RoboDK station: Drillingtask2.rdk

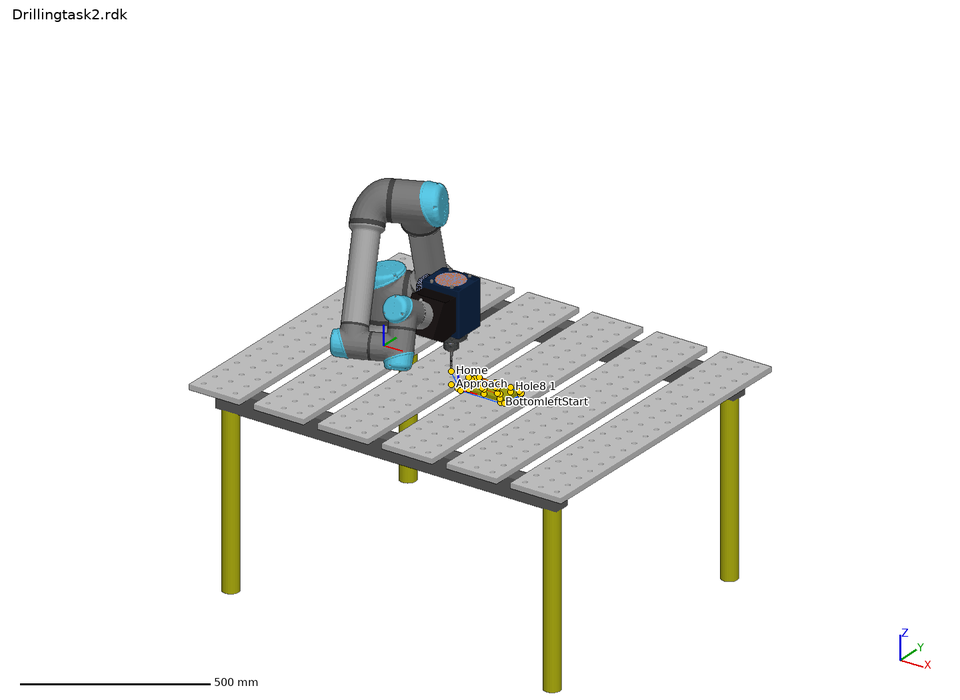
[picture v0: the station drawn from its stored meshes, robots at their saved joint values, targets as dots, program paths as lines]
Station Drillingtask2 (saved by RoboDK 5.6.3). Poses are relative to the parent item; angles as X-Y-Z fixed-axis rotations.
  - frame UR5e Base at (0, 0, 0) mm
    - robot UR5e: 6 axes, payload 5 kg, reach 850 mm, repeatability 0.03 mm, weight 18.4 kg
        modified DH rows (alpha deg, a mm, theta deg, d mm): 0, 0, 0, 162.5; 90, 0, 180, 0; 0, 425, 0, 0; 0, 392.25, 0, 133.3; -90, 0, 0, 99.7; 90, 0, 180, 99.6
        joint limits [-360, -360, -360, -360, -360, -360] to [360, 360, 360, 360, 360, 360]; home [0, -90, -90, 0, 90, 0]; saved at [113.645, -60.354, -246.748, 94.881, 69.676, 12.348]
      - tool Custom Spindle, TCP at (0, 119.5, 220.16) mm, rotated rx -60 ry 0 rz 0 deg, size 260.9 x 152 x 222 mm, geometry from Custom Spindle.STEP
  - object Object Table at (310, 0, 0) mm, size 1193.8 x 965.2 x 609.6 mm, geometry from Object Table.wrl
  - frame Frame 2 at (310, -100, 0) mm
    - object Drilling_Part at (0, 0, 0) mm, size 150 x 75 x 10 mm, geometry from Part2.sld
    - target Home  (Cartesian target) at (-30, 10, 40) mm, rotated rx -180 ry 0 rz 0 deg; joints [113.645, -60.354, -246.748, 94.881, 69.676, 12.348] of UR5e
    - target Approach (Cartesian target) at (-30, 10, 0) mm, rotated rx 180 ry 0 rz 0 deg; joints [113.645, -55.5, -246.2, 89.479, 69.676, 12.348] of UR5e
    - folder Side
      - target TopleftStart (Cartesian target) at (-4, 10, 0) mm, rotated rx -180 ry 0 rz 0 deg; joints [116.986, -54.016, -249.586, 90.663, 66.86, 14.284] of UR5e
      - target TopLeftCorner (Cartesian target) at (0, 0, 0) mm, rotated rx 180 ry 0 rz 0 deg; joints [116.854, -53.181, -251.371, 91.644, 66.971, 14.206] of UR5e
      - target TopleftAfter (Cartesian target) at (10, -4, 0) mm, rotated rx 180 ry 0 rz 0 deg; joints [117.797, -52.339, -253.229, 92.437, 66.18, 14.766] of UR5e
      - target BottomleftStart (Cartesian target) at (140, -4, 0) mm, rotated rx 180 ry 0 rz 0 deg; joints [130.532, -43.004, -273.82, 99.603, 55.75, 23.148] of UR5e
      - target BottomleftCorner (Cartesian target) at (150, 0, 0) mm, rotated rx 180 ry 0 rz 0 deg; joints [131.612, -42.384, -275.208, 99.917, 54.893, 23.946] of UR5e
      - target BottomleftFinish (Cartesian target) at (154, 10, 0) mm, rotated rx -180 ry 0 rz 0 deg; joints [132.635, -42.601, -274.851, 99.328, 54.085, 24.719] of UR5e
      - target BottomrightStart (Cartesian target) at (154, 65, 0) mm, rotated rx -180 ry 0 rz 0 deg; joints [136.857, -45.391, -269.503, 94.72, 50.81, 28.08] of UR5e
      - target Bottomrightcorner (Cartesian target) at (150, 75, 0) mm, rotated rx -180 ry 0 rz 0 deg; joints [137.377, -46.192, -267.904, 93.645, 50.413, 28.516] of UR5e
      - target BottomrightAfter (Cartesian target) at (140, 79, 0) mm, rotated rx 180 ry 0 rz 0 deg; joints [136.932, -47.226, -265.698, 92.71, 50.753, 28.142] of UR5e
      - target ToprightStart (Cartesian target) at (10, 79, 0) mm, rotated rx 180 ry 0 rz 0 deg; joints [123.819, -56.892, -243.887, 85.983, 61.184, 18.519] of UR5e
      - target ToprightCorner (Cartesian target) at (0, 75, 0) mm, rotated rx 180 ry 0 rz 0 deg; joints [122.196, -57.332, -242.797, 85.825, 62.521, 17.475] of UR5e
      - target ToprightFinish (Cartesian target) at (-4, 65, 0) mm, rotated rx 180 ry 0 rz 0 deg; joints [120.864, -57.071, -243.255, 86.401, 63.623, 16.637] of UR5e
    - target ApproachDrill (Cartesian target) at (25, 12.5, 35) mm, rotated rx -180 ry 0 rz 0 deg; joints [120.595, -56.265, -253.761, 96.175, 63.847, 16.47] of UR5e
    - folder Folder 2
      - target Hole1 1 (Cartesian target) at (25, 12.5, 15) mm, rotated rx 180 ry 0 rz 0 deg; joints [120.595, -54.074, -253.452, 93.676, 63.847, 16.47] of UR5e
      - target Hole1 2 (Cartesian target) at (25, 12.5, 1) mm, rotated rx -180 ry 0 rz 0 deg; joints [120.595, -52.494, -253.321, 91.965, 63.847, 16.47] of UR5e
      - target Hole1 3 (Cartesian target) at (25, 12.5, 15) mm, rotated rx 180 ry 0 rz 0 deg; joints [120.595, -54.074, -253.452, 93.676, 63.847, 16.47] of UR5e
      - target Hole2 1 (Cartesian target) at (75, 12.5, 15) mm, rotated rx -180 ry 0 rz 0 deg; joints [125.89, -50.54, -261.032, 96.097, 59.49, 19.89] of UR5e
      - target Hole2 2 (Cartesian target) at (75, 12.5, 1) mm, rotated rx -180 ry 0 rz 0 deg; joints [125.89, -49.093, -260.897, 94.515, 59.49, 19.89] of UR5e
      - target Hole2 3 (Cartesian target) at (75, 12.5, 15) mm, rotated rx -180 ry 0 rz 0 deg; joints [125.89, -50.54, -261.032, 96.097, 59.49, 19.89] of UR5e
      - target Hole3 1 (Cartesian target) at (125, 12.5, 15) mm, rotated rx -180 ry 0 rz 0 deg; joints [130.456, -46.595, -269.436, 98.841, 55.81, 23.093] of UR5e
      - target Hole3 2 (Cartesian target) at (125, 12.5, 1) mm, rotated rx -180 ry 0 rz 0 deg; joints [130.456, -45.268, -269.294, 97.372, 55.81, 23.093] of UR5e
      - target Hole3 3 (Cartesian target) at (125, 12.5, 15) mm, rotated rx -180 ry 0 rz 0 deg; joints [130.456, -46.595, -269.436, 98.841, 55.81, 23.093] of UR5e
      - target Hole4 1 (Cartesian target) at (100, 37.5, 15) mm, rotated rx 180 ry 0 rz 0 deg; joints [130.121, -49.997, -262.491, 95.434, 56.078, 22.848] of UR5e
      - target Hole4 2 (Cartesian target) at (100, 37.5, 1) mm, rotated rx 180 ry 0 rz 0 deg; joints [130.121, -48.576, -262.349, 93.871, 56.078, 22.848] of UR5e
      - target Hole4 3 (Cartesian target) at (100, 37.5, 15) mm, rotated rx 180 ry 0 rz 0 deg; joints [130.121, -49.997, -262.491, 95.434, 56.078, 22.848] of UR5e
      - target Hole5 1 (Cartesian target) at (50, 37.5, 15) mm, rotated rx -180 ry 0 rz 0 deg; joints [125.155, -53.78, -254.375, 92.927, 60.089, 19.399] of UR5e
      - target Hole5 2 (Cartesian target) at (50, 37.5, 1) mm, rotated rx 180 ry 0 rz 0 deg; joints [125.155, -52.221, -254.238, 91.23, 60.089, 19.399] of UR5e
      - target Hole5 3 (Cartesian target) at (50, 37.5, 15) mm, rotated rx -180 ry 0 rz 0 deg; joints [125.155, -53.78, -254.375, 92.927, 60.089, 19.399] of UR5e
      - target Hole6 1 (Cartesian target) at (25, 62.5, 15) mm, rotated rx -180 ry 0 rz 0 deg; joints [124.29, -56.901, -247.952, 89.907, 60.797, 18.827] of UR5e
      - target Hole6 2 (Cartesian target) at (25, 62.5, 1) mm, rotated rx 180 ry 0 rz 0 deg; joints [124.29, -55.211, -247.811, 88.076, 60.797, 18.827] of UR5e
      - target Hole6 3 (Cartesian target) at (25, 62.5, 15) mm, rotated rx -180 ry 0 rz 0 deg; joints [124.29, -56.901, -247.952, 89.907, 60.797, 18.827] of UR5e
      - target Hole7 1 (Cartesian target) at (75, 62.5, 15) mm, rotated rx -180 ry 0 rz 0 deg; joints [129.732, -53.24, -255.873, 92.216, 56.389, 22.567] of UR5e
      - target Hole7 2 (Cartesian target) at (75, 62.5, 1) mm, rotated rx -180 ry 0 rz 0 deg; joints [129.732, -51.711, -255.728, 90.543, 56.389, 22.567] of UR5e
      - target Hole7 3 (Cartesian target) at (75, 62.5, 15) mm, rotated rx -180 ry 0 rz 0 deg; joints [129.732, -53.24, -255.873, 92.216, 56.389, 22.567] of UR5e
      - target Hole8 1 (Cartesian target) at (125, 62.5, 15) mm, rotated rx 180 ry 0 rz 0 deg; joints [134.319, -49.211, -264.507, 94.816, 52.768, 26.024] of UR5e
      - target Hole8 2 (Cartesian target) at (125, 62.5, 1) mm, rotated rx -180 ry 0 rz 0 deg; joints [134.319, -47.823, -264.356, 93.277, 52.768, 26.024] of UR5e
      - target Hole8 3 (Cartesian target) at (125, 62.5, 15) mm, rotated rx 180 ry 0 rz 0 deg; joints [134.319, -49.211, -264.507, 94.816, 52.768, 26.024] of UR5e
  - program Home (3 instructions, listed below)
  - program Approach (3 instructions, listed below)
  - program Side (12 instructions, listed below)
  - program Home (3 instructions, listed below)
  - program Approachdrill (3 instructions, listed below)
  - program Drilling (26 instructions, listed below)
  - program Home (3 instructions, listed below)
  - program SideAndDrill (7 instructions, listed below)
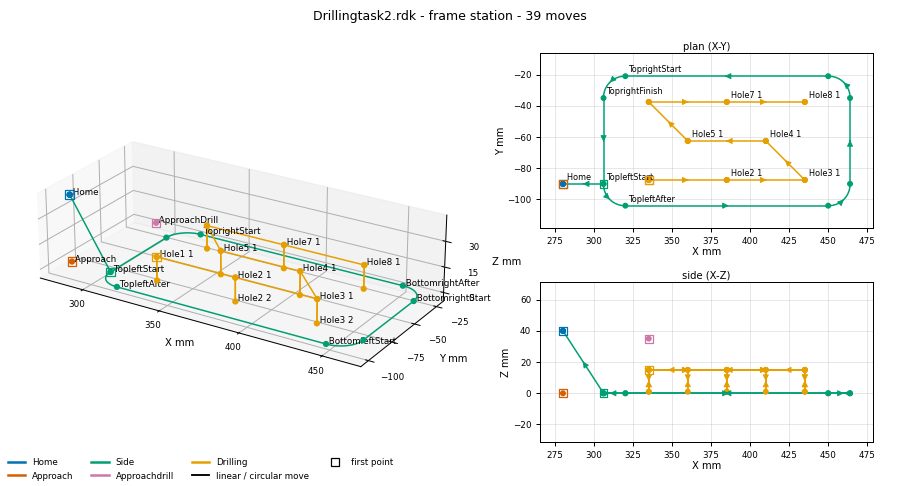
[picture p0: tool path of Drillingtask2.rdk in frame station, 39 of 39 moves have a stored position in this frame; points joined in program order, loops and branches not executed]

--- program Home (robot UR5e) ---
  Set Ref.: Frame 2
  Set Tool: Custom Spindle
  MoveL (Home )

--- program Approach (robot UR5e) ---
  Set Ref.: Frame 2
  Set Tool: Custom Spindle
  MoveL (Approach)

--- program Side (robot UR5e) ---
  Set Ref.: Frame 2
  Set Tool: Custom Spindle
  MoveL (TopleftStart)
  MoveC (TopLeftCorner, TopleftAfter)
  MoveL (BottomleftStart)
  MoveC (BottomleftCorner, BottomleftFinish)
  MoveL (BottomrightStart)
  MoveC (Bottomrightcorner, BottomrightAfter)
  MoveL (ToprightStart)
  MoveC (ToprightCorner, ToprightFinish)
  MoveL (TopleftStart)
  MoveL (Home )

--- program Home (robot UR5e) ---
  Set Ref.: Frame 2
  Set Tool: Custom Spindle
  MoveL (Home )

--- program Approachdrill (robot UR5e) ---
  Set Ref.: Frame 2
  Set Tool: Custom Spindle
  MoveL (ApproachDrill)

--- program Drilling (robot UR5e) ---
  Set Ref.: Frame 2
  Set Tool: Custom Spindle
  MoveL (Hole1 1)
  MoveL (Hole1 2)
  MoveL (Hole1 3)
  MoveL (Hole2 1)
  MoveL (Hole2 2)
  MoveL (Hole2 3)
  MoveL (Hole3 1)
  MoveL (Hole3 2)
  MoveL (Hole3 3)
  MoveL (Hole4 1)
  MoveL (Hole4 2)
  MoveL (Hole4 3)
  MoveL (Hole5 1)
  MoveL (Hole5 2)
  MoveL (Hole5 3)
  MoveL (Hole6 1)
  MoveL (Hole6 2)
  MoveL (Hole6 3)
  MoveL (Hole7 1)
  MoveL (Hole7 2)
  MoveL (Hole7 3)
  MoveL (Hole8 1)
  MoveL (Hole8 2)
  MoveL (Hole8 3)

--- program Home (robot UR5e) ---
  Set Ref.: Frame 2
  Set Tool: Custom Spindle
  MoveL (Home )

--- program SideAndDrill (robot UR5e) ---
  Call Home
  Call Approach
  Call Side
  Call Home
  Call Approachdrill
  Call Drilling
  Call Home
